PROGRAM ReactorFlowController
VAR_INPUT
	serialCommData : ST_SerialCommReadData;
	flowControlValveOpening : DINT;
	serialCommReadData : ST_SerialCommReadData;
END_VAR
VAR
	
	// Handlers to call
	HandleCo2MeanFlowCalculation : FB_Co2MeanFlowCalculationHandler;
	HandleCo2Consumption : FB_Co2consumptionHandler;
	HandleCo2FlowModeling : FB_Co2FlowModelingHandler;
	HandleCo2FlowModelDeviation : FB_Co2FlowModelDeviationHandler(maxValue := 0.35);
	HandleFlowMpc : FB_FlowMpcHandler;
	
	// Local variables
	_meanReactorFlow : REAL;
	_flowControlParameters : ST_FlowControlParameters;
	_consumedCo2Amount : REAL;
	_flowControlCommands : ST_FlowControlCommands;
	_co2ConsumptionLimitExceeded : BOOL;
	_modeledReactorMeanFlow : REAL;
	_closeOnOffValve : BOOL;
	_flowModelDeviationPercentage : DINT;
END_VAR

HandleCo2MeanFlowCalculation(
				serialCommData := serialCommData,
				flowControlParameters := _flowControlParameters,
				startCalculation := _flowControlCommands.startMovingAvgCalculation,
				meanReactorFlow => _meanReactorFlow);
				
HandleCo2Consumption(
				meanFlow := _meanReactorFlow,
				flowControlParameters := _flowControlParameters,
				resetInput := _flowControlCommands.resetCo2Consumption,
				consumedCo2Amount => _consumedCo2Amount,
				limitExceeded => _co2ConsumptionLimitExceeded,
				closeOnOffValve => _closeOnOffValve);
				
HandleCo2FlowModeling(
				valvePositionPercentage := flowControlValveOpening,
				pumpingPressureDelta := serialCommReadData.pumpingPressureSetpoint-serialCommReadData.pumpingPressureMeasurement,
				flowMeasurement := _meanReactorFlow,
				modelingActive := _flowControlCommands.startMovingAvgCalculation,
				modeledOutput => _modeledReactorMeanFlow);
				
HandleCo2FlowModelDeviation(
				currentFlow := _meanReactorFlow,
				modeledFlow := _modeledReactorMeanFlow,
				deviationPercentage => _flowModelDeviationPercentage);
				
HandleFlowMpc(
			flowSetpoint := ,
			pumpingPressureDelta := serialCommReadData.pumpingPressureSetpoint-serialCommReadData.pumpingPressureMeasurement,
			currentValvePosition := ReactorLevelAndPressureController.ControlValveOpening,
			modeledValvePercentage := ,
			flowModel := HandleCo2FlowModeling.mF);

PROPERTY CloseOnOffValve : BOOL
GET

CloseOnOffValve := _closeOnOffValve;
END_GET
END_PROPERTY

PROPERTY Co2ConsumptionLimitExceeded : BOOL
GET

Co2ConsumptionLimitExceeded := _co2ConsumptionLimitExceeded;
END_GET
END_PROPERTY

PROPERTY ConsumedCo2Amount : REAL
GET

ConsumedCo2Amount := _consumedCo2Amount;
END_GET
END_PROPERTY

PROPERTY FlowControlCommands : ST_FlowControlCommands
SET

_flowControlCommands := FlowControlCommands;
END_SET
END_PROPERTY

PROPERTY FlowControlParameters : ST_FlowControlParameters
SET

_flowControlParameters := FlowControlParameters;
END_SET
END_PROPERTY

PROPERTY FlowModelDeviationPercentage : DINT
GET

FlowModelDeviationPercentage := _flowModelDeviationPercentage;
END_GET
END_PROPERTY

PROPERTY MeanReactorFlow : REAL
GET

MeanReactorFlow := _meanReactorFlow;
END_GET
END_PROPERTY

PROPERTY ModeledMeanReactorFlow : REAL
GET

ModeledMeanReactorFlow := _modeledReactorMeanFlow;
END_GET
END_PROPERTY

END_PROGRAM

(* stored: Version 1.1.0.1, ProductVersion 3.1.4024.9
   POU ReactorFlowController: Id {610f8bfd-64ff-403d-a02a-9c006717ec6e}, SpecialFunc None
   Property CloseOnOffValve: Id {f2106895-29cc-4255-a249-f7d05f58ca87}
   Get Get: Id {0fcd2bfe-a430-4321-886c-289ced6cc77c}
   Property Co2ConsumptionLimitExceeded: Id {e63d7dc5-de1e-4e21-892b-686d47b989ed}
   Get Get: Id {f79d35cf-ce48-4946-856f-8b1a17ac789d}
   Property ConsumedCo2Amount: Id {15d55ab9-92af-4bd7-9af9-6676fe5e9820}
   Get Get: Id {7cb71c26-fc41-4127-ad9c-30da31ebea17}
   Property FlowControlCommands: Id {06bb8475-5eea-42cb-9fdb-40ae1ea8f78d}
   Set Set: Id {f79b2c5f-cdd2-4a83-8b38-9e3160ac7049}
   Property FlowControlParameters: Id {3952f682-48f7-4a6b-97c4-f9cb206094ff}
   Set Set: Id {bb7ee2b7-b99b-4b22-a116-ec0a74f99722}
   Property FlowModelDeviationPercentage: Id {22a43f75-ad1c-4ffc-94e5-2f0f90ba56e2}
   Get Get: Id {3d84f36f-90b5-441d-b9fe-9d60886be910}
   Property MeanReactorFlow: Id {54cf3119-bfc4-4992-9290-14785dcc2c4c}
   Get Get: Id {d74e12b3-eeff-426f-95ec-b4d7bd07139c}
   Property ModeledMeanReactorFlow: Id {d89940c1-e57b-4ab0-80d4-4a5c5dd1e9d7}
   Get Get: Id {1d1f071e-5a92-4ab8-b188-21226a15a07f} *)
